Fanuc KAREL source: kt00520.KL

PROGRAM KT00520
%STACKSIZE=65535
%PRIORITY=65535
%NOLOCKGROUP
VAR
P1 : XYZWPREXT
P2 : XYZWPR
OUT : XYZWPR
BEGIN
P1.X=1.0
P2.Y=2.0
-- UNRESOLVED_PC line 10 opcodes [49 7E 49 7E 60 7E 4A] marker_code=40
END KT00520
